FUNCTION_BLOCK FB_Generator IMPLEMENTS IGenerator
VAR_INPUT
END_VAR
VAR_OUTPUT
END_VAR
VAR
	ton1		:TON;
	tCycleTime		:TIME;
	bBlink			:BOOL;
END_VAR

{warning 'add method implementation'}
METHOD Flash : BOOL
ton1(IN:=NOT ton1.Q, PT:= tCycleTime, Q=> , ET=> );

IF	ton1.Q THEN 
	bBlink := NOT bBlink;
END_IF

Flash	:= bBlink;
END_METHOD

{warning 'add property implementation'}
PROPERTY P_tCycleTime : TIME
GET
P_tCycleTime := tCycleTime;
END_GET
SET
tCycleTime := P_tCycleTime;
END_SET
END_PROPERTY

{warning 'add property implementation'}
PROPERTY P_Vendor : STRING
GET
P_Vendor := 'Google';
END_GET
END_PROPERTY

END_FUNCTION_BLOCK

(* stored: Version 1.1.0.1, ProductVersion 3.1.4022.16
   POU FB_Generator: Id {9e09a7b5-ff34-4256-969c-0d7828266939}, SpecialFunc None
   Method Flash: Id {abc50991-7468-4d97-aff4-e20ac3d116d5}
   Property P_tCycleTime: Id {e425694d-87cf-4ce8-8500-a30ad0ed0e54}
   Get Get: Id {5dd535b9-3bb1-4256-97ab-6ed36a6ea0c9}
   Set Set: Id {6643e2ce-cb44-4158-aa48-fc2806f0bab8}
   Property P_Vendor: Id {d36f3d71-11a1-4f50-b724-def219d7641f}
   Get Get: Id {df1d1215-3a27-472a-8d64-165c63b1d955} *)
